{attribute 'GeneratedUsingTerminal: EL6861-0000-0016'}
{attribute addProperty BoxType "EL6861-0000-0016"}
{attribute addProperty Id "Transmit_requestBOOL1Receive_acceptedBOOL1Init_requestBOOL1Send_continuousBOOL1Output_lenUSINT1"}
{attribute addProperty CRC "3864532377"}
{attribute addProperty Size "5"}
TYPE Ctrl_E6581599 :
STRUCT
	{attribute addProperty Name "Transmit_request"}
	Transmit_request : BOOL;
	{attribute addProperty Name "Receive_accepted"}
	Receive_accepted : BOOL;
	{attribute addProperty Name "Init_request"}
	Init_request : BOOL;
	{attribute addProperty Name "Send_continuous"}
	Send_continuous : BOOL;
	{attribute addProperty Name "Output_len"}
	Output_len : USINT;
END_STRUCT
END_TYPE

(* stored: Version 1.2.0.0, ProductVersion 3.1.4024.11
   DUT Ctrl_E6581599: Id {3ffceac6-4500-46cc-9c54-ca3d68eb9f1f} *)
